FUNCTION_BLOCK XtsIoEnvVar IMPLEMENTS I_XtsIoEnvVar, I_Object, I_Initialisable
VAR
	XtsIoEnvironment : Tc3_XTS_Utility.FB_TcIoXtsEnvironment;
	stXtsEnvironmentConfiguration	: ST_XtsEnvironmentConfiguration;
	_Initialised : BOOL;
END_VAR

METHOD FB_init : BOOL
VAR_INPUT
	bInitRetains : BOOL; // if TRUE, the retain variables are initialized (warm start / cold start)
	bInCopyCode : BOOL;  // if TRUE, the instance afterwards gets moved into the copy code (online change)
END_VAR
stXtsEnvironmentConfiguration.bEnableInitCaGroup := TRUE;
XtsIoEnvironment.P_XtsEnvironmentConfiguration := stXtsEnvironmentConfiguration;
END_METHOD

METHOD GetCaGroupInterface : I_Mc2CaGroup
VAR_INPUT
	CAGroupNumber : INT;
END_VAR
IF NOT Initialised THEN
	RETURN;
END_IF

GetCaGroupInterface := XtsIoEnvironment.Mc2CaGroup(TO_UINT(CAGroupNumber));
END_METHOD

METHOD GetXPUInterface : I_TcIoXtsProcessingUnit
VAR_INPUT
	MyXts : INT;
END_VAR
IF NOT Initialised THEN
	RETURN;
END_IF

GetXPUInterface := XtsIoEnvironment.XpuTcIo(TO_UINT(MyXts));
END_METHOD

METHOD PUBLIC Initialise : HRESULT
VAR_INPUT
END_VAR
IF XtsIoEnvironment.Init(TRUE) THEN
	XtsIoEnvironment.Init(FALSE);
	_Initialised := TRUE;
ELSE
	Initialise := -1;
END_IF
END_METHOD

PROPERTY Initialised : BOOL
GET
Initialised := _Initialised;
END_GET
END_PROPERTY

METHOD RegisterWithParent
VAR_INPUT
	Parent	: I_HostObjects;
END_VAR
Parent.RegisterInitialisable(THIS^);
END_METHOD

END_FUNCTION_BLOCK

(* stored: Version 1.1.0.1
   POU XtsIoEnvVar: Id {03c3c931-6ee3-4ab9-88b9-320f3e1d8e15}, SpecialFunc None
   Folder Commands: Id {3a159131-d61b-452b-8e2f-6ee920e4571d}
   Folder Status: Id {11c58542-69d8-416b-8e98-b88ed835287f}
   Method FB_init: Id {5798f5d6-785a-4124-98b0-b4ab031dfdac}
   Method GetCaGroupInterface: Id {12f834a0-9ae6-48b5-9bae-7bc717cd2b2d}
   Method GetXPUInterface: Id {a6b4198a-d372-4fc0-b700-debb44563dc0}
   Method Initialise: Id {f0d17991-21f7-403c-899a-0fcccbff041e}
   Property Initialised: Id {0f4a9fc3-49d6-473e-a6e3-78db8cfcf818}
   Get Get: Id {820b3227-250d-444d-bfaf-048041bb942e}
   Method RegisterWithParent: Id {37203846-0f41-471d-b37e-9d946dd0bd38} *)
